FUNCTION_BLOCK InputChannelV2BOOL (* Basic Function Block Type *)
  (* Standard: 61499-2 *)
  (* Version 0.0, 12/03/2018, Atmojo, nxtControl GmbH, Template *)
  PACKAGE Main;
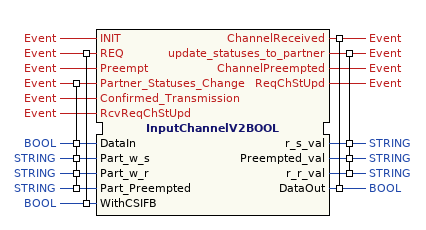
  EVENT_INPUT
    INIT;
    REQ WITH WithCSIFB; (* Normal Execution Request *)
    Preempt;
    Partner_Statuses_Change WITH DataIn, Part_w_s, Part_w_r, Part_Preempted;
    Confirmed_Transmission;
    RcvReqChStUpd;
  END_EVENT
  EVENT_OUTPUT
    ChannelReceived WITH DataOut; (* Execution Confirmation *)
    update_statuses_to_partner WITH r_s_val, Preempted_val, r_r_val;
    ChannelPreempted;
    ReqChStUpd;
  END_EVENT
  VAR_INPUT
    DataIn : BOOL;
    Part_w_s : STRING;
    Part_w_r : STRING;
    Part_Preempted : STRING;
    WithCSIFB : BOOL;
  END_VAR
  VAR_OUTPUT
    r_s_val : STRING := '0';
    Preempted_val : STRING := '0';
    r_r_val : STRING := '0';
    DataOut : BOOL;
  END_VAR
  VAR
    Part_w_s_localcopy : INT := 0;
    Part_w_r_localcopy : INT := 0;
    Part_preempted_localcopy : INT := 0;
    r_s : INT := 0;
    r_r : INT := 0;
    data_buffer : BOOL;
    Chan_Preempted_Status : INT := 0;
    reqCount : INT := 0;
    ChanIsUsed : BOOL := FALSE;
    WithCSIFBStat : BOOL := FALSE;
  END_VAR
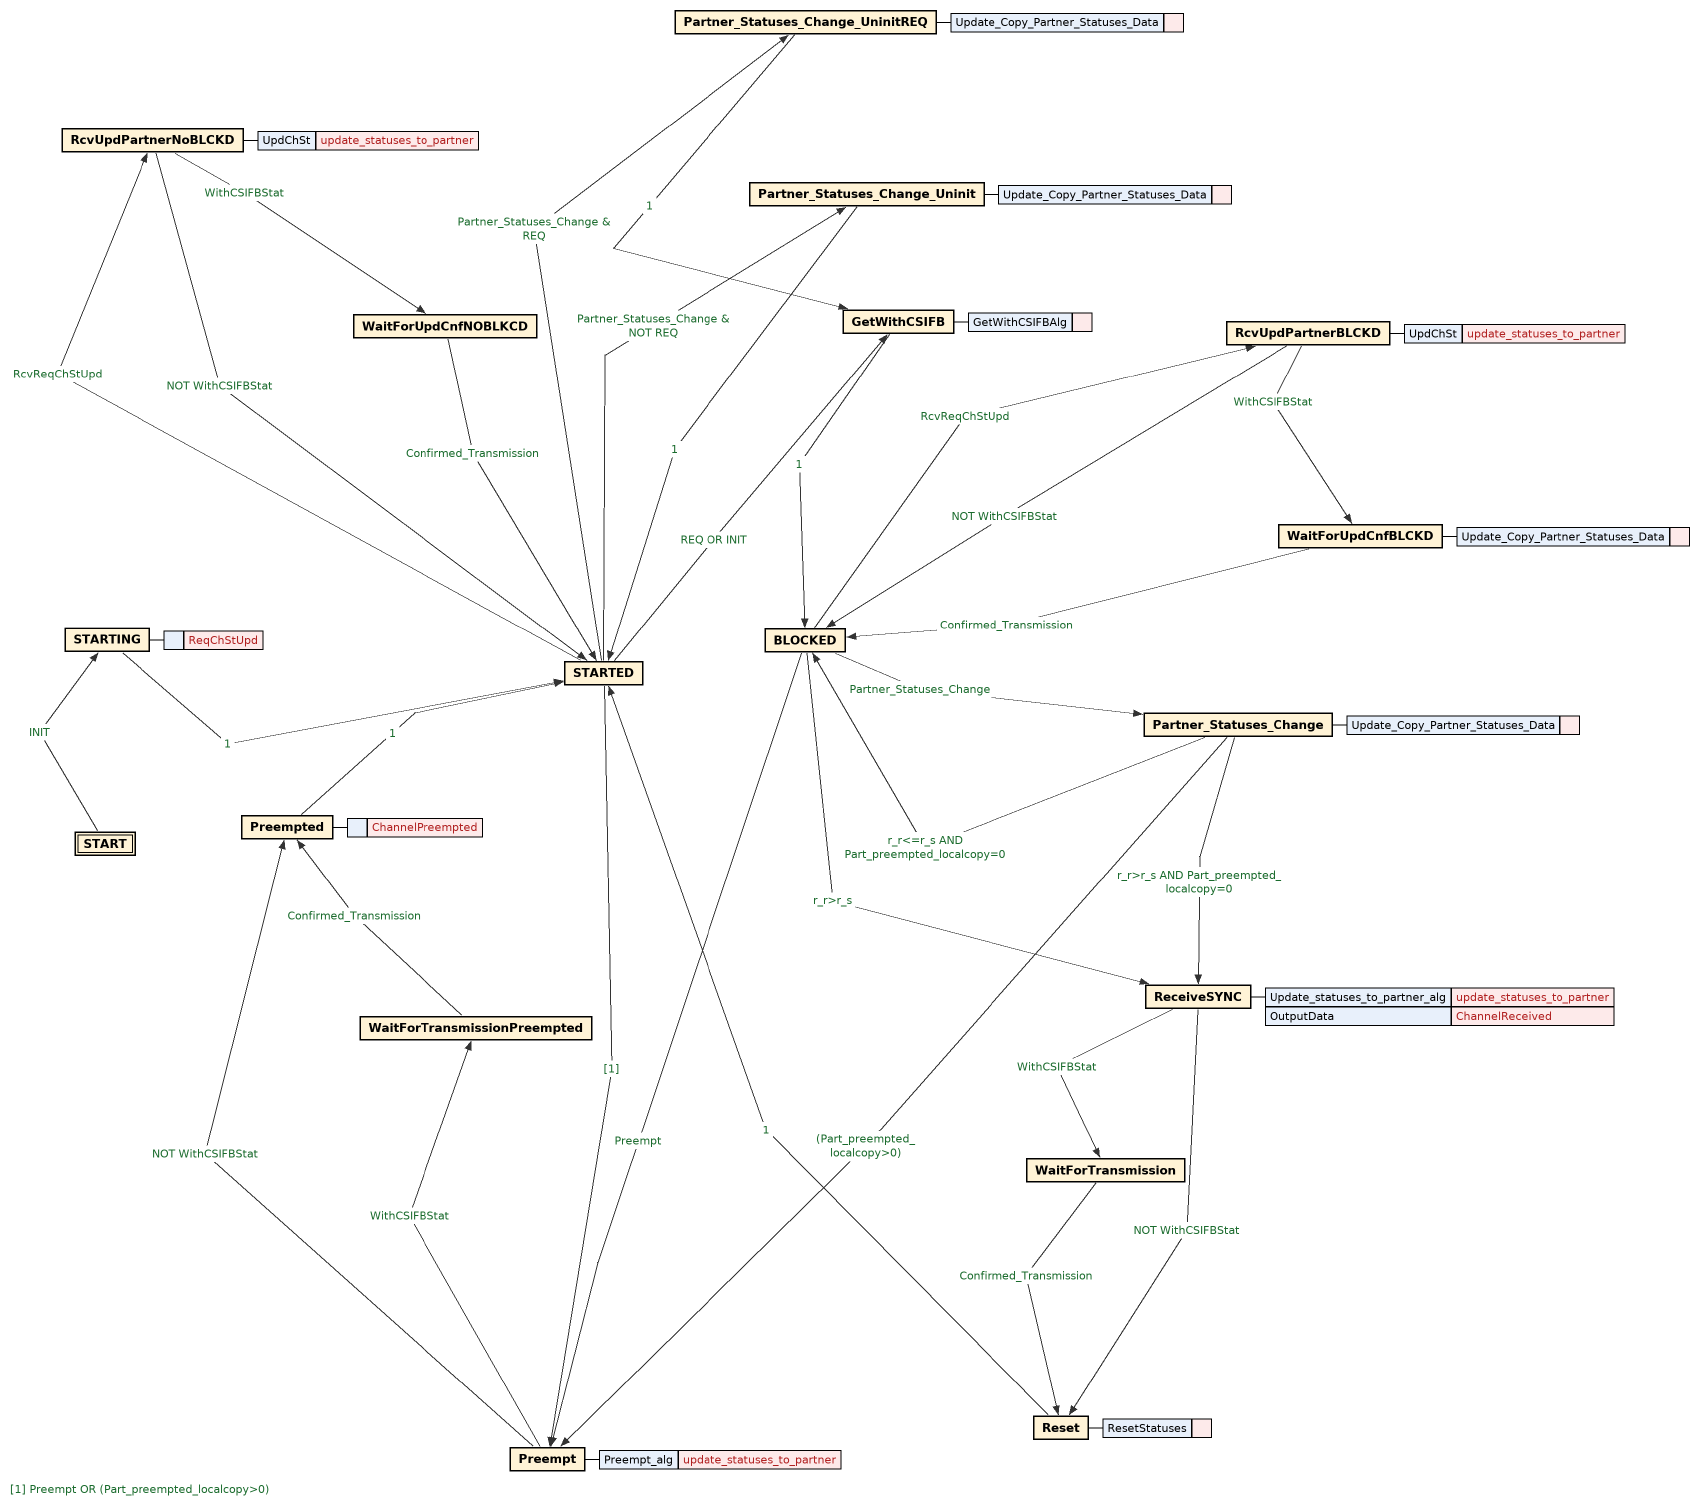
  EC_STATES
    START; (* Initial State *)
    Preempt : Preempt_alg -> update_statuses_to_partner;
    BLOCKED;
    Partner_Statuses_Change : Update_Copy_Partner_Statuses_Data;
    ReceiveSYNC : Update_statuses_to_partner_alg -> update_statuses_to_partner, OutputData -> ChannelReceived;
    Partner_Statuses_Change_Uninit : Update_Copy_Partner_Statuses_Data;
    WaitForTransmission;
    WaitForTransmissionPreempted;
    Preempted : -> ChannelPreempted;
    GetWithCSIFB : GetWithCSIFBAlg;
    STARTING : -> ReqChStUpd;
    STARTED;
    RcvUpdPartnerNoBLCKD : UpdChSt -> update_statuses_to_partner;
    RcvUpdPartnerBLCKD : UpdChSt -> update_statuses_to_partner;
    WaitForUpdCnfNOBLKCD;
    WaitForUpdCnfBLCKD : Update_Copy_Partner_Statuses_Data;
    Partner_Statuses_Change_UninitREQ : Update_Copy_Partner_Statuses_Data;
    Reset : ResetStatuses;
  END_STATES
  EC_TRANSITIONS
    STARTED TO Preempt := Preempt OR (Part_preempted_localcopy>0);
    WaitForTransmissionPreempted TO Preempted := Confirmed_Transmission;
    BLOCKED TO Preempt := Preempt;
    BLOCKED TO Partner_Statuses_Change := Partner_Statuses_Change;
    Partner_Statuses_Change TO ReceiveSYNC := r_r>r_s AND Part_preempted_localcopy=0;
    Partner_Statuses_Change TO BLOCKED := r_r<=r_s AND Part_preempted_localcopy=0;
    Partner_Statuses_Change TO Preempt := (Part_preempted_localcopy>0);
    STARTED TO Partner_Statuses_Change_Uninit := Partner_Statuses_Change & NOT REQ;
    Partner_Statuses_Change_Uninit TO STARTED := 1;
    ReceiveSYNC TO WaitForTransmission := WithCSIFBStat;
    Preempt TO WaitForTransmissionPreempted := WithCSIFBStat;
    Preempted TO STARTED := 1;
    WaitForTransmission TO Reset := Confirmed_Transmission;
    STARTED TO GetWithCSIFB := REQ OR INIT;
    BLOCKED TO ReceiveSYNC := r_r>r_s;
    ReceiveSYNC TO Reset := NOT WithCSIFBStat;
    Preempt TO Preempted := NOT WithCSIFBStat;
    GetWithCSIFB TO BLOCKED := 1;
    START TO STARTING := INIT;
    STARTING TO STARTED := 1;
    STARTED TO RcvUpdPartnerNoBLCKD := RcvReqChStUpd;
    RcvUpdPartnerNoBLCKD TO STARTED := NOT WithCSIFBStat;
    BLOCKED TO RcvUpdPartnerBLCKD := RcvReqChStUpd;
    RcvUpdPartnerBLCKD TO BLOCKED := NOT WithCSIFBStat;
    RcvUpdPartnerNoBLCKD TO WaitForUpdCnfNOBLKCD := WithCSIFBStat;
    WaitForUpdCnfNOBLKCD TO STARTED := Confirmed_Transmission;
    RcvUpdPartnerBLCKD TO WaitForUpdCnfBLCKD := WithCSIFBStat;
    WaitForUpdCnfBLCKD TO BLOCKED := Confirmed_Transmission;
    STARTED TO Partner_Statuses_Change_UninitREQ := Partner_Statuses_Change & REQ;
    Partner_Statuses_Change_UninitREQ TO GetWithCSIFB := 1;
    Reset TO STARTED := 1;
  END_TRANSITIONS
  ALGORITHM Preempt_alg IN ST:
r_s:=0;
r_r:=0;

r_r_val:=INT_TO_STRING (r_r);
r_s_val:=INT_TO_STRING (r_s);
Preempted_val:=INT_TO_STRING (Chan_Preempted_Status+1);
  END_ALGORITHM
  ALGORITHM Update_Copy_Partner_Statuses_Data IN ST:
Part_w_r_localcopy:=STRING_TO_INT(Part_w_r);
Part_w_s_localcopy:=STRING_TO_INT(Part_w_s);
Part_preempted_localcopy:=STRING_TO_INT(Part_Preempted);
data_buffer:=DataIn;
r_r:=Part_w_s_localcopy;
r_s:=Part_w_r_localcopy;
  END_ALGORITHM
  ALGORITHM Update_Copy_Partner_Preempted_Status IN ST:
Part_preempted_localcopy:=STRING_TO_INT(Part_Preempted);
  END_ALGORITHM
  ALGORITHM Update_statuses_to_partner_alg IN ST:
r_s:=r_s+1;
r_s_val:=INT_TO_STRING (r_s);
r_r_val:=INT_TO_STRING (r_r);
Preempted_val:= INT_TO_STRING (Chan_Preempted_Status);
  END_ALGORITHM
  ALGORITHM ResetStatuses IN ST:
data_buffer:=FALSE;
DataOut:=FALSE;
r_s:=0;
r_r:=0;
Chan_Preempted_Status:=0;
Part_preempted_localcopy:=0;
r_r_val:='0';
r_s_val:='0';
Preempted_val:='0';
  END_ALGORITHM
  ALGORITHM GetWithCSIFBAlg IN ST:
WithCSIFBStat:=WithCSIFB;
  END_ALGORITHM
  ALGORITHM UpdChSt IN ST:
r_s_val:=INT_TO_STRING (r_s);
r_r_val:=INT_TO_STRING (r_r);
Preempted_val:= INT_TO_STRING (Chan_Preempted_Status);
  END_ALGORITHM
  ALGORITHM OutputData IN ST:
DataOut:=data_buffer;
  END_ALGORITHM
END_FUNCTION_BLOCK
